// TIA Portal V19 export
FUNCTION_BLOCK "TYPIC_C904_IF_VPI"   // FB37, FBD
TITLE = TYPIC_C904_IF_VPI: Vuilvloeistof
{ S7_Optimized_Access := 'TRUE' }
AUTHOR : OCOTECH
FAMILY : Typical
NAME : C904.702
// Logisch Object Besturing: C904.702
// 
// De interne functie vuilvloeistof verzorgt de algemene handbediening via een aanraakscherm.
// stored: MemoryReserve 10, SetENOAutomatically false
   VAR_OUTPUT
      VAR_IF_VPI { ExternalAccessible := 'False'; ExternalVisible := 'False'; ExternalWritable := 'False'} : "C904_VAR_IF_VPI_TYPIC";   // Struct met alle variabelen naar bovenliggende functies
   END_VAR
   VAR_IN_OUT
      STU_IF_VPI : USInt;   // Gewenst regime
   END_VAR
   VAR
      BED : Struct   // Bedieningen
         AFSTAND : Bool;   // Bediening om pompinstallatie in afstand te schakelen
         LOZ : Bool;   // Bediening om pompinstallatie in regime Lozen te schakelen
         UIT : Bool;   // Bediening om pompinstallatie in regime Uit te schakelen
      END_STRUCT;
      VAR { ExternalWritable := 'False'} : Struct   // Variabelen
         WRE : USInt;   // Actueel actief regime
         BMO_HAND : Bool;   // TRUE = Regime handmatig ingesteld via lokale bediening
      END_STRUCT;
   END_VAR
BEGIN

REGION Network 1: START
END_REGION

REGION Network 2: +++ Bepalen regime en bedieningsmode +++
   // Actueel regime via handbediening instellen en bepalen van de bedieningsmode HAND.
END_REGION

REGION Network 3 (SCL): EINDE
   // Variabelen van intern scada rakvlak naar outputs copieren
   #VAR_IF_VPI.WRE := #VAR.WRE;
   #VAR_IF_VPI.BMO_HAND := #VAR.BMO_HAND;
END_REGION
END_FUNCTION_BLOCK
